FUNCTION_BLOCK FB_A10
VAR_INPUT
END_VAR
VAR_OUTPUT
END_VAR
VAR
END_VAR

METHOD M_reset : BOOL
VAR_INPUT
END_VAR
//////////////////////reset all error here////////////////////////////
END_METHOD

END_FUNCTION_BLOCK

(* stored: Version 1.1.0.1, ProductVersion 3.1.4024.12
   POU FB_A10: Id {61bf9701-30d1-49ea-a466-b92010020989}, SpecialFunc None
   Method M_reset: Id {29fb3e66-dea3-478b-9f0c-92be7a310a7e} *)
